(* Specifies the direction of a ramping signal. *)
{attribute 'qualified_only'}
{attribute 'strict'}
{attribute 'to_string'}
TYPE E_RampDirection :
(
	Rising   := 0, // Output increases over time.
	Falling  := 1  // Output decreases over time.
)BYTE;
END_TYPE

(* stored: Version 1.1.0.1, ProductVersion 3.1.4024.15
   EnumerationTextList E_RampDirection: Id {4711f057-537b-4304-ad1b-cbfea61da026} *)
